// Layout checklist: REFERENCE TO is an address, not the referent.
// Kept apart from ST_PointerWidth so that a compiler which refuses a
// REFERENCE member inside a STRUCT costs this rule alone.
TYPE ST_ReferenceWidth :
STRUCT
	leadIn : BYTE;
	target : REFERENCE TO INT;
	trailer : BYTE;
END_STRUCT
END_TYPE

(* stored: Version 1.1.0.1, ProductVersion 3.1.4026.18
   DUT ST_ReferenceWidth: Id {c0de1a70-0000-4000-8000-000000000002} *)
